TYPE Block64Words :
UNION
	reserved : ARRAY[1..64] OF WORD; //memeory occupation
	axis : AxisBase;
	//cylinder : cylinderBlockBase;
	signal : signalBlockbase;
	command : commandBlockGeneric;
	unit : UnitBase;
END_UNION
END_TYPE

(* stored: Version 1.1.0.1, ProductVersion 3.1.4022.10
   DUT Block64Words: Id {45a09079-c4b6-4675-89db-e70c1695c394} *)
